FUNCTION_BLOCK FB_Button
VAR_INPUT
	bButtonPress : BOOL;
END_VAR
VAR_OUTPUT
	nCounter: INT;
END_VAR
VAR
END_VAR

END_FUNCTION_BLOCK

(* stored: Version 1.1.0.1
   POU FB_Button: Id {6d28b3f1-4f56-4f8c-bdc4-881946647258}, SpecialFunc None *)
